FUNCTION_BLOCK CmdVentValvesBasic (* Basic Function Block Type *)
  (* Standard: 61499-2 *)
  (* Version 0.0, 8/9/2024, SESA713705, Schneider Electric, Template *)
  PACKAGE SE.Nereda;
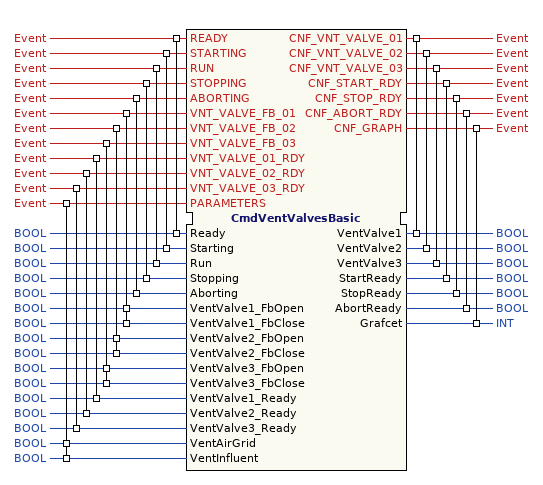
  EVENT_INPUT
    READY WITH Ready;
    STARTING WITH Starting;
    RUN WITH Run;
    STOPPING WITH Stopping;
    ABORTING WITH Aborting;
    VNT_VALVE_FB_01 WITH VentValve1_FbOpen, VentValve1_FbClose;
    VNT_VALVE_FB_02 WITH VentValve2_FbOpen, VentValve2_FbClose;
    VNT_VALVE_FB_03 WITH VentValve3_FbOpen, VentValve3_FbClose;
    VNT_VALVE_01_RDY WITH VentValve1_Ready;
    VNT_VALVE_02_RDY WITH VentValve2_Ready;
    VNT_VALVE_03_RDY WITH VentValve3_Ready;
    PARAMETERS WITH VentAirGrid, VentInfluent;
  END_EVENT
  EVENT_OUTPUT
    CNF_VNT_VALVE_01 WITH VentValve1;
    CNF_VNT_VALVE_02 WITH VentValve2;
    CNF_VNT_VALVE_03 WITH VentValve3;
    CNF_START_RDY WITH StartReady;
    CNF_STOP_RDY WITH StopReady;
    CNF_ABORT_RDY WITH AbortReady;
    CNF_GRAPH WITH Grafcet;
  END_EVENT
  VAR_INPUT
    Ready : BOOL;
    Starting : BOOL;
    Run : BOOL;
    Stopping : BOOL;
    Aborting : BOOL;
    VentValve1_FbOpen : BOOL;
    VentValve1_FbClose : BOOL;
    VentValve2_FbOpen : BOOL;
    VentValve2_FbClose : BOOL;
    VentValve3_FbOpen : BOOL;
    VentValve3_FbClose : BOOL;
    VentValve1_Ready : BOOL;
    VentValve2_Ready : BOOL;
    VentValve3_Ready : BOOL;
    VentAirGrid : BOOL;
    VentInfluent : BOOL;
  END_VAR
  VAR_OUTPUT
    VentValve1 : BOOL; (* Vent Air Grid Valve : NVPP 001 a—036 *)
    VentValve2 : BOOL; (* NVPP 001 a—038 *)
    VentValve3 : BOOL; (* Vent Influent Valve : NVPP 001 a—067 *)
    StartReady : BOOL;
    StopReady : BOOL;
    AbortReady : BOOL;
    Grafcet : INT;
  END_VAR
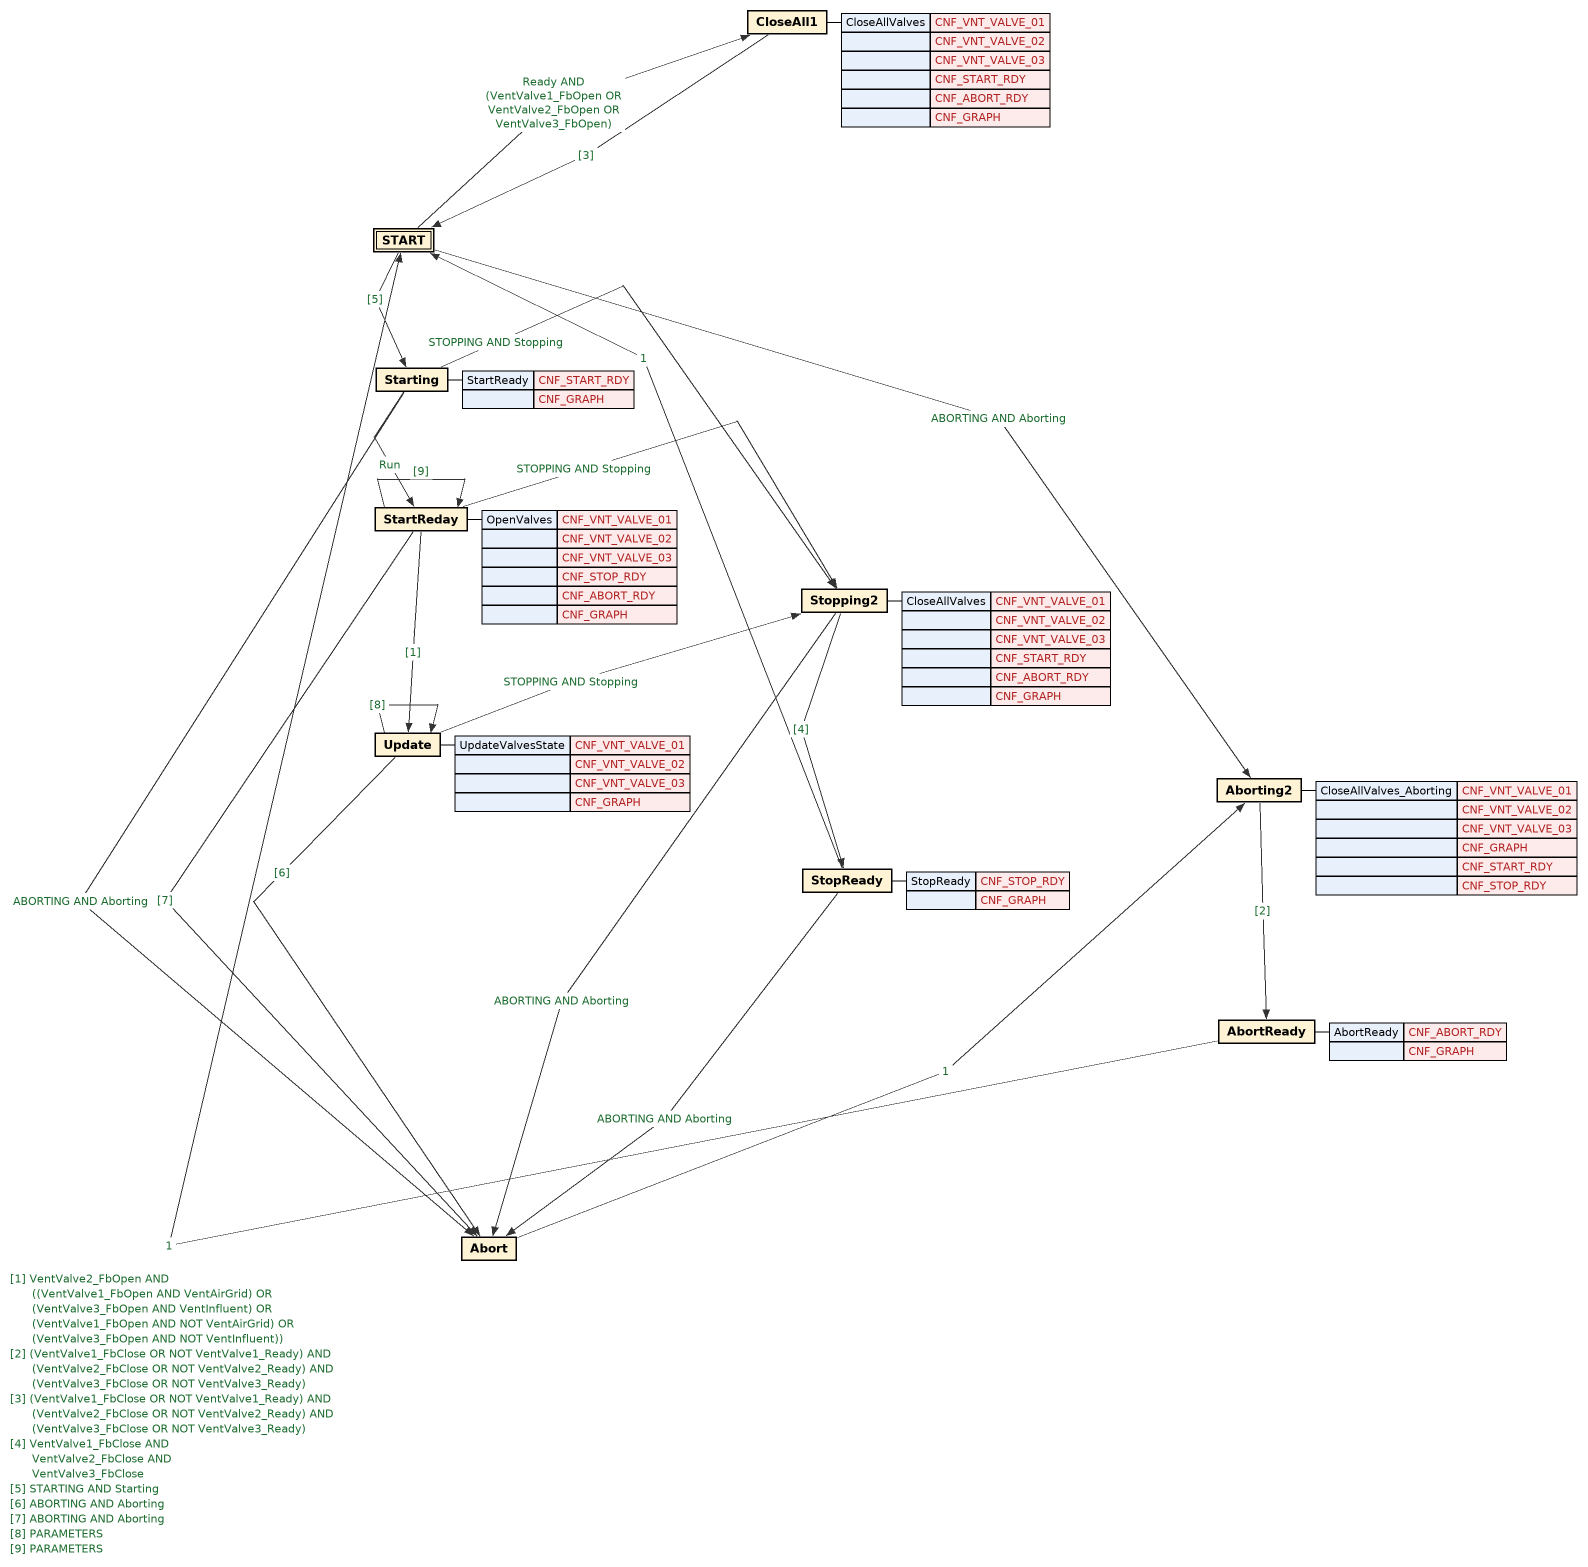
  EC_STATES
    START; (* Initial State *)
    Starting : StartReady -> CNF_START_RDY, -> CNF_GRAPH;
    Abort;
    StopReady : StopReady -> CNF_STOP_RDY, -> CNF_GRAPH;
    Update : UpdateValvesState -> CNF_VNT_VALVE_01, -> CNF_VNT_VALVE_02, -> CNF_VNT_VALVE_03, -> CNF_GRAPH;
    AbortReady : AbortReady -> CNF_ABORT_RDY, -> CNF_GRAPH;
    StartReday : OpenValves -> CNF_VNT_VALVE_01, -> CNF_VNT_VALVE_02, -> CNF_VNT_VALVE_03, -> CNF_STOP_RDY, -> CNF_ABORT_RDY, -> CNF_GRAPH;
    Aborting2 : CloseAllValves_Aborting -> CNF_VNT_VALVE_01, -> CNF_VNT_VALVE_02, -> CNF_VNT_VALVE_03, -> CNF_GRAPH, -> CNF_START_RDY, -> CNF_STOP_RDY;
    Stopping2 : CloseAllValves -> CNF_VNT_VALVE_01, -> CNF_VNT_VALVE_02, -> CNF_VNT_VALVE_03, -> CNF_START_RDY, -> CNF_ABORT_RDY, -> CNF_GRAPH;
    CloseAll1 : CloseAllValves -> CNF_VNT_VALVE_01, -> CNF_VNT_VALVE_02, -> CNF_VNT_VALVE_03, -> CNF_START_RDY, -> CNF_ABORT_RDY, -> CNF_GRAPH;
  END_STATES
  EC_TRANSITIONS
    START TO CloseAll1 := Ready AND (VentValve1_FbOpen OR VentValve2_FbOpen OR VentValve3_FbOpen);
    START TO Starting := STARTING AND Starting;
    Update TO Stopping2 := STOPPING AND Stopping;
    START TO Aborting2 := ABORTING AND Aborting;
    Starting TO StartReday := Run;
    Abort TO Aborting2 := 1;
    Update TO Update := PARAMETERS;
    Stopping2 TO Abort := ABORTING AND Aborting;
    Starting TO Abort := ABORTING AND Aborting;
    Update TO Abort := ABORTING AND Aborting;
    Aborting2 TO AbortReady := (VentValve1_FbClose OR NOT VentValve1_Ready) AND (VentValve2_FbClose OR NOT VentValve2_Ready) AND (VentValve3_FbClose OR NOT VentValve3_Ready);
    StopReady TO Abort := ABORTING AND Aborting;
    AbortReady TO START := 1;
    StopReady TO START := 1;
    Stopping2 TO StopReady := VentValve1_FbClose AND VentValve2_FbClose AND VentValve3_FbClose;
    CloseAll1 TO START := (VentValve1_FbClose OR NOT VentValve1_Ready) AND (VentValve2_FbClose OR NOT VentValve2_Ready) AND (VentValve3_FbClose OR NOT VentValve3_Ready);
    StartReday TO StartReday := PARAMETERS;
    StartReday TO Update := VentValve2_FbOpen AND ((VentValve1_FbOpen AND VentAirGrid) OR (VentValve3_FbOpen AND VentInfluent) OR (VentValve1_FbOpen AND NOT VentAirGrid) OR (VentValve3_FbOpen AND NOT VentInfluent));
    StartReday TO Stopping2 := STOPPING AND Stopping;
    StartReday TO Abort := ABORTING AND Aborting;
    Starting TO Stopping2 := STOPPING AND Stopping;
  END_TRANSITIONS
  ALGORITHM CloseAllValves IN ST:
;

VentValve1 := FALSE;
VentValve2 := FALSE;
VentValve3 := FALSE;

StartReady := FALSE;
AbortReady := FALSE;
  END_ALGORITHM
  ALGORITHM StartReady IN ST:
;
Grafcet := 2;
StartReady := TRUE;
  END_ALGORITHM
  ALGORITHM OpenValves IN ST:
;
//VentValve1 : NVPP 001 a—036
//VentValve2 : NVPP 001 a—038
//VentValve3 : NVPP 001 a—067

Grafcet := 2;
StopReady := FALSE;
AbortReady := FALSE;
VentValve2 := TRUE;

IF NOT VentAirGrid AND NOT VentInfluent THEN
	VentValve1 := FALSE;
	VentValve3 := FALSE;

ELSIF VentAirGrid AND NOT VentInfluent THEN
	VentValve1 := TRUE;
	VentValve3 := FALSE;

ELSIF NOT VentAirGrid AND VentInfluent THEN
	VentValve1 := FALSE;
	VentValve3 := TRUE;

ELSIF VentAirGrid AND VentInfluent THEN
	VentValve1 := TRUE;
	VentValve3 := TRUE;
END_IF;
  END_ALGORITHM
  ALGORITHM UpdateValvesState IN ST:
;
//VentValve1 : NVPP 001 a—036
//VentValve2 : NVPP 001 a—038
//VentValve3 : NVPP 001 a—067

Grafcet := 4;
VentValve2 := TRUE;

IF NOT VentAirGrid AND NOT VentInfluent THEN
	VentValve1 := FALSE;
	VentValve3 := FALSE;

ELSIF VentAirGrid AND NOT VentInfluent THEN
	VentValve1 := TRUE;
	VentValve3 := FALSE;

ELSIF NOT VentAirGrid AND VentInfluent THEN
	VentValve1 := FALSE;
	VentValve3 := TRUE;

ELSIF VentAirGrid AND VentInfluent THEN
	VentValve1 := TRUE;
	VentValve3 := TRUE;
END_IF;
  END_ALGORITHM
  ALGORITHM AbortReady IN ST:
;
Grafcet := 10;
AbortReady := TRUE;
  END_ALGORITHM
  ALGORITHM StopReady IN ST:
;
Grafcet := 7;
StopReady := TRUE;
  END_ALGORITHM
  ALGORITHM StopBlowers_WhenAborting IN ST:
;
StartReady := FALSE;
StopReady := FALSE;
  END_ALGORITHM
  ALGORITHM CloseAllValves_Aborting IN ST:
;
VentValve1 := FALSE;
VentValve2 := FALSE;
VentValve3 := FALSE;

StartReady := FALSE;
StopReady := FALSE;
  END_ALGORITHM
END_FUNCTION_BLOCK
